{attribute 'linkalways'} 
{attribute 'no_explicit_call' := 'This FB is a CLASS and must be accessed using methods or properties'}
{attribute 'enable_dynamic_creation'}
FUNCTION_BLOCK _ETcVnDistanceTransformationMask EXTENDS EnumDatatypeBase
VAR
	localData : ETcVnDistanceTransformationMask;
	activeData : REFERENCE TO ETcVnDistanceTransformationMask;
	enumBaseDatatype : _DINT(localData);
END_VAR

METHOD PRIVATE AddLocalEnumeration
VAR_INPUT
	Enumeration : T_MAXSTRING;
	Value : ETcVnDistanceTransformationMask;
END_VAR
AddEnumeration(Enumeration, Value);
END_METHOD

PROPERTY PUBLIC Address : PVOID
GET
Address := ADR(activeData);
END_GET
END_PROPERTY

METHOD PUBLIC ClearReference
VAR_INPUT
END_VAR
activeData REF= localData;
SetBaseDatatypeReference();
END_METHOD

METHOD PUBLIC Clone : I_Datatype
VAR
    pClone : POINTER TO _ETcVnDistanceTransformationMask;
END_VAR
pClone := __NEW(_ETcVnDistanceTransformationMask(InitialValue := Value));
Clone := pClone^;
END_METHOD

METHOD FB_init : BOOL
VAR_INPUT
	bInitRetains : BOOL; // if TRUE, the retain variables are initialized (warm start / cold start)
	bInCopyCode : BOOL;  // if TRUE, the instance afterwards gets moved into the copy code (online change)
	InitialValue : ETcVnDistanceTransformationMask;
END_VAR
localData := InitialValue;
AddBaseDatatype(enumBaseDatatype);
ClearReference();

AddLocalEnumeration('TCVN_DTM_PRECISE', ETcVnDistanceTransformationMask.TCVN_DTM_PRECISE);
AddLocalEnumeration('TCVN_DTM_3', ETcVnDistanceTransformationMask.TCVN_DTM_3);
AddLocalEnumeration('TCVN_DTM_5', ETcVnDistanceTransformationMask.TCVN_DTM_5);
END_METHOD

PROPERTY PUBLIC Identifier : T_MAXSTRING
GET
Identifier := 'ETcVnDistanceTransformationMask';
END_GET
END_PROPERTY

METHOD IsEnumeratorValueEqual : BOOL
VAR_INPUT
	Enumerator : I_KeyValueForwardEnumerator;
END_VAR
VAR
	storedValue : ETcVnDistanceTransformationMask;
END_VAR
IF NOT Enumerator.TryGet(storedValue) THEN
	RETURN;
END_IF

IsEnumeratorValueEqual := storedValue = activeData;
END_METHOD

METHOD PUBLIC MakeReferenceTo
VAR_INPUT
	ReferenceTarget : REFERENCE TO ETcVnDistanceTransformationMask;
END_VAR
activeData REF= ReferenceTarget;
SetBaseDatatypeReference();
END_METHOD

METHOD PROTECTED SetBaseDatatypeReference
VAR_INPUT
END_VAR
enumBaseDatatype.MakeReferenceTo(activeData);
END_METHOD

PROPERTY PUBLIC Size : UDINT
GET
Size := SIZEOF(activeData);
END_GET
END_PROPERTY

METHOD TryMakeReferenceTo : BOOL
VAR_INPUT
	Target : I_Datatype;
END_VAR
VAR
	targetAsEnum : I_EnumDatatype;
	pTargetData : POINTER TO ETcVnDistanceTransformationMask;
END_VAR
IF NOT Target.TryResolveAsEnumDatatype(targetAsEnum) THEN
	RETURN;
END_IF

IF targetAsEnum.Identifier <> Identifier THEN
	RETURN;
END_IF

pTargetData := Target.Address;
activeData REF= pTargetData^;
SetBaseDatatypeReference();
TryMakeReferenceTo := TRUE;
END_METHOD

PROPERTY PUBLIC Value : ETcVnDistanceTransformationMask
GET
Value := activeData;
END_GET
SET
activeData := Value;
END_SET
END_PROPERTY

END_FUNCTION_BLOCK

(* stored: Version 1.1.0.1, ProductVersion 3.1.4024.13
   POU _ETcVnDistanceTransformationMask: Id {4cec14f4-7ded-0f53-2dcf-7d1ce37b04ee}, SpecialFunc None
   Folder Core: Id {9ec177de-771d-012b-08c4-a3408966bf57}
   Folder Protected: Id {abe7bdb4-9b2a-074f-2be2-92c01cbe5b7f}
   Folder Customize: Id {f9bf7d00-d009-0f02-00d5-5ab85117b5e0}
   Folder Constructor: Id {c8016806-f6de-0e86-0d68-07ae249b5bb6}
   Folder Private: Id {907fcd79-eedc-0a05-1697-00f30a678ef6}
   Folder Protected: Id {a10f5122-f8ca-0402-3e98-e3105066a3aa}
   Method AddLocalEnumeration: Id {d3e106b1-d56b-07da-137e-311c6ee8fa96}
   Property Address: Id {cc25bdfd-bd1d-0156-106e-57f6366e5d70}
   Get Get: Id {ef3b2dbb-d518-03bf-2f69-feb977487d2b}
   Method ClearReference: Id {0b116283-b83d-0eae-34fd-b4e71b80d983}
   Method Clone: Id {a0b3ca03-9a0e-066b-2c88-08c113ad6feb}
   Method FB_init: Id {b6c1a8c2-f47c-0786-2ccd-224d4f2918d6}
   Property Identifier: Id {6582ca6b-b45b-025d-1c25-7f31e69c44ee}
   Get Get: Id {2df06628-c1a5-0b4e-154c-40792bc40b4b}
   Method IsEnumeratorValueEqual: Id {4a83dbcc-e881-0cf5-092e-c5c012ab8ac2}
   Method MakeReferenceTo: Id {9c39befc-32ba-0001-0781-dde2ffa73397}
   Method SetBaseDatatypeReference: Id {20aa3484-903b-010f-04a1-d8e6b7743ff7}
   Property Size: Id {b8214e5a-fdb8-09a2-324f-aba1f2567b25}
   Get Get: Id {bda5b24c-48eb-00fd-1d00-2ca2e5a85f37}
   Method TryMakeReferenceTo: Id {477f2439-0551-0893-3d67-e379d1d8340d}
   Property Value: Id {102934ec-41c0-066f-34ba-f9ae308b500a}
   Get Get: Id {1d2d76a7-a88a-0449-3ee6-f39c9b4f840a}
   Set Set: Id {bab1d74e-67bc-0357-1f84-20d32d2c2df0} *)
